// TIA Portal V17 export
// export: Created 2025-03-07T09:17:02.3863953Z, ExportSetting WithDefaults, DisplayName Totally Integrated Automation Portal, DisplayVersion V17 Update 8, DisplayName TIA Portal Openness, DisplayVersion V17 Update 8, DisplayName TIA Portal Version Control Interface, DisplayVersion V17, DisplayName SINAMICS Startdrive Advanced, DisplayVersion V17 SP2, DisplayName SINAMICS Startdrive G110M, G120, G120C, G120D, G120P, G115D, DisplayVersion V17 SP2, DisplayName SINAMICS Startdrive G130, G150, S120, S150, SINAMICS MV, S210, DisplayVersion V17 SP2, DisplayName STEP 7 Professional, DisplayVersion V17 Update 8, DisplayName SINUMERIK ONE STEP 7 Toolbox, DisplayVersion V17 Update 12, DisplayName SINUMERIK 840D sl STEP 7 Toolbox, DisplayVersion V17 Update 12, DisplayName STEP 7 Safety, DisplayVersion V17 Update 6, DisplayName WinCC Advanced, DisplayVersion V17 Update 8
DATA_BLOCK "DB7300_INTERLOCK_GENERAL"   // DB7300
{ S7_Optimized_Access := 'FALSE'; DB_Accessible_From_OPC_UA := 'FALSE' }
AUTHOR : ETXETAR
VERSION : 1.0
// stored: AutoNumber false, DBAccessibleFromOPCUA false, DBAccessibleFromWebserver true, IsOnlyStoredInLoadMemory false, IsWriteProtectedInAS false
   VAR RETAIN
      GENERAL_MACHINE : Struct
         FROM_CELL_TO_MACHINE_GENERAL : Struct
            CELL_MEAS_STA_START_CYCLE : Bool;   // CELL MEASURING STATION START CYCLE
            CELL_MEAS_STA_CALIB_CYCLE : Bool;   // CELL MEASURING STATION CALIBRATION CYCLE
            CELL_MEAS_STA_HOME_REQ : Bool;   // CELL MEASURING STATION HOME REQUEST
            CELL_MEAS_STA_FAULT : Bool;   // CELL MEASURING STATION FAULT
            CELL_MEAS_STA_RESET : Bool;   // CELL MEASURING STATION RESET
            CALIB_MODE_SLCTD_TEMP : Bool;   // CALIBRATION MODE SELECTED TEMP
            CELL_COOLING_DEGRADED_MODE : Bool;   // CELL COOLING DEGRADED MODE
            CELL_STARVED : Bool;   // CELL STARVED
            CELL_BLOCKED : Bool;   // CELL BLOCKED
         END_STRUCT;
         FROM_ROBOT_TO_UNIT_01 : Struct
            HEARTBEAT : Bool;   // ROBOT HEARTBEAT
            EMERG_STOP_OK : Bool;   // ROBOT EMERGENCY STOP OK
            ROBOT_FAULT : Bool;   // ROBOT FAULT
            SAFETY_DOOR_CLSD_LOCKD : Bool;   // ROBOT SAFETY DOOR CLOSED AND LOCKED
            CELL_EMPTY : Bool;   // ROBOT CELL EMPTY
            IN_MANUAL_MODE : Bool;   // ROBOT MANUAL MODE SELECTED
            IN_AUTO_MODE : Bool;   // ROBOT AUTO MODE SELECTED
            IN_AUTO_CYCLE_RUN : Bool;   // ROBOT CYCLE RUNNING IN AUTOMATIC MODE
            RUN_OUT_REQUEST : Bool;   // ROBOT MACHINE RUN OUT REQUEST
            RUN_OUT_COMPLETED : Bool;   // ROBOT RUN OUT COMPLETED
            SAFETY_DOOR_OPEN_REQ : Bool;   // ROBOT ANY CELL SAFETY DOOR OPEN REQUEST
            OK_TO_OPEN_SAFETY_GATES : Bool;   // OK TO OPEN SAFETY GATES
            READY_TO_SERVICE : Bool;   // ROBOT READY TO SERVICE MACHINE
            OUT_OF_COLLISION_MACHINE : Bool;   // ROBOT OUT OF COLLISION MACHINE
            OUT_OF_COLLISION_FIXTURE : Bool;   // ROBOT OUT OF COLLISION FIXTURE
            PART_ENABLED : Bool;   // ROBOT PART ENABLED
            PART_FACE_R_TO_DELIVER : Bool;   // ROBOT PART FACE R TO DELIVER IMMEDIATELY
            PART_FACE_N_TO_DELIVER : Bool;   // ROBOT PART FACE N TO DELIVER IMMEDIATELY
            OUT_OF_PARTS_FACE_R_TO_DELIVER : Bool;   // ROBOT OUT OF PARTS FACE R IN CELL TO DELIVER
            OUT_OF_PARTS_FACE_N_TO_DELIVER : Bool;   // ROBOT OUT OF PARTS FACE N IN CELL TO DELIVER
            PART_LOADED : Bool;   // ROBOT PART LOADED
            PART_UNLOADED : Bool;   // ROBOT PART UNLOADED
            FIX_SKIP_REQ : Bool;   // ROBOT FIXTURE SKIP REQUEST
            PART_TYPE_CHANGE_REQ : Bool;   // ROBOT PART TYPE CHANGE REQUEST
            PART_TYPE : Byte;   // ROBOT PART TYPE
         END_STRUCT;
         FROM_ROBOT_TO_UNIT_02 : Struct
            HEARTBEAT : Bool;   // ROBOT HEARTBEAT
            EMERG_STOP_OK : Bool;   // ROBOT EMERGENCY STOP OK
            ROBOT_FAULT : Bool;   // ROBOT FAULT
            SAFETY_DOOR_CLSD_LOCKD : Bool;   // ROBOT SAFETY DOOR CLOSED AND LOCKED
            CELL_EMPTY : Bool;   // ROBOT CELL EMPTY
            IN_MANUAL_MODE : Bool;   // ROBOT MANUAL MODE SELECTED
            IN_AUTO_MODE : Bool;   // ROBOT AUTO MODE SELECTED
            IN_AUTO_CYCLE_RUN : Bool;   // ROBOT CYCLE RUNNING IN AUTOMATIC MODE
            RUN_OUT_REQUEST : Bool;   // ROBOT MACHINE RUN OUT REQUEST
            RUN_OUT_COMPLETED : Bool;   // ROBOT RUN OUT COMPLETED
            SAFETY_DOOR_OPEN_REQ : Bool;   // ROBOT ANY CELL SAFETY DOOR OPEN REQUEST
            OK_TO_OPEN_SAFETY_GATES : Bool;   // OK TO OPEN SAFETY GATES
            READY_TO_SERVICE : Bool;   // ROBOT READY TO SERVICE MACHINE
            OUT_OF_COLLISION_MACHINE : Bool;   // ROBOT OUT OF COLLISION MACHINE
            OUT_OF_COLLISION_FIXTURE : Bool;   // ROBOT OUT OF COLLISION FIXTURE
            PART_ENABLED : Bool;   // ROBOT PART ENABLED
            PART_FACE_R_TO_DELIVER : Bool;   // ROBOT PART FACE R TO DELIVER IMMEDIATELY
            PART_FACE_N_TO_DELIVER : Bool;   // ROBOT PART FACE N TO DELIVER IMMEDIATELY
            OUT_OF_PARTS_FACE_R_TO_DELIVER : Bool;   // ROBOT OUT OF PARTS FACE R IN CELL TO DELIVER
            OUT_OF_PARTS_FACE_N_TO_DELIVER : Bool;   // ROBOT OUT OF PARTS FACE N IN CELL TO DELIVER
            PART_LOADED : Bool;   // ROBOT PART LOADED
            PART_UNLOADED : Bool;   // ROBOT PART UNLOADED
            FIX_SKIP_REQ : Bool;   // ROBOT FIXTURE SKIP REQUEST
            PART_TYPE_CHANGE_REQ : Bool;   // ROBOT PART TYPE CHANGE REQUEST
            PART_TYPE : Byte;   // ROBOT PART TYPE
         END_STRUCT;
      END_STRUCT;
      POWDER_PLC : Struct
         GENERAL : Struct
            LIFE_BIT : Bool;   // LIFE BIT
            SELECTED_ARGON_GAS : Bool;   // SELECTED ARGON GAS
            SELECTED_NITROGEN_GAS : Bool;   // SELECTED NITROGEN GAS
            SELECTED_IMPERIAL_SYSTEM : Bool;   // SELECTED IMPERIAL SYSTEM
            SELECTED_METRIC_SYSTEM : Bool;   // SELECTED METRIC SYSTEM
            POWDER_PLC_AUTO_MODE : Bool;   // POWDER PLC IN AUTO MODE
            POWDER_PLC_MAN_MODE : Bool;   // POWDER PLC IN MANUAL MODE
         END_STRUCT;
         FROM_POWDER_TO_UNIT_01 : Struct
            POWDER_UNIT_01_READY_TO_RUN : Bool;   // POWDER UNIT 01 READY TO RUN
            POWDER_UNIT_01_STOPPED : Bool;   // POWDER UNIT 01 STOPPED
            SWITCHED_ON_POWDER_UNIT_01 : Bool;   // SWITCHED ON POWDER UNIT 01
            SWITCHED_OFF_POWDER_UNIT_01 : Bool;   // SWITCHED OFF POWDER UNIT 01
            SWITCHED_ON_TEMPERATURE_JACKET_UNIT_01 : Bool;   // SWITCHED ON TEMPERATURE JACKET UNIT 01
            SWITCHED_OFF_TEMPERATURE_JACKET_UNIT_01 : Bool;   // SWITCHED OFF TEMPERATURE JACKET UNIT 01
            POWDER_UNIT_01_ALARM : Bool;   // POWDER UNIT 01 ALARM
            UNIT_01_POWDER_FEEDER_1_CARRIER_GAS_ACTUAL_LINE_1 : Real;   // UNIT 01 POWDER FEEDER 1 CARRIER GAS ACTUAL LINE 1
            UNIT_01_POWDER_FEEDER_1_DISK_SPEED_ACTUAL_LINE_1 : Real;   // UNIT 01 POWDER FEEDER 1 DISK SPEED ACTUAL LINE 1
            UNIT_01_POWDER_FEEDER_1_STIRRER_SPEED_ACTUAL_LINE_1 : Real;   // UNIT 01 POWDER FEEDER 1 STIRRER SPEED ACTUAL LINE 1
            UNIT_01_POWDER_FEEDER_1_HOPPER_TEMPERATURE_ACTUAL_LINE_1 : Real;   // UNIT 01 POWDER FEEDER 1 HOPPER TEMPERATURE ACTUAL LINE 1
            UNIT_01_POWDER_FEEDER_1_CARRIER_GAS_ACTUAL_LINE_2 : Real;   // UNIT 01 POWDER FEEDER 1 CARRIER GAS ACTUAL LINE 2
            UNIT_01_POWDER_FEEDER_1_DISK_SPEED_ACTUAL_LINE_2 : Real;   // UNIT 01 POWDER FEEDER 1 DISK SPEED ACTUAL LINE 2
            UNIT_01_POWDER_FEEDER_1_STIRRER_SPEED_ACTUAL_LINE_2 : Real;   // UNIT 01 POWDER FEEDER 1 STIRRER SPEED ACTUAL LINE 2
            UNIT_01_POWDER_FEEDER_1_HOPPER_TEMPERATURE_ACTUAL_LINE_2 : Real;   // UNIT 01 POWDER FEEDER 1 HOPPER TEMPERATURE ACTUAL LINE 2
         END_STRUCT;
         FROM_POWDER_TO_UNIT_02 : Struct
            POWDER_UNIT_02_READY_TO_RUN : Bool;   // POWDER UNIT 02 READY TO RUN
            POWDER_UNIT_02_STOPPED : Bool;   // POWDER UNIT 02 STOPPED
            SWITCHED_ON_POWDER_UNIT_02 : Bool;   // SWITCHED ON POWDER UNIT 02
            SWITCHED_OFF_POWDER_UNIT_02 : Bool;   // SWITCHED OFF POWDER UNIT 02
            SWITCHED__ON_TEMPERATURE_JACKET_UNIT_02 : Bool;   // SWITCHED ON TEMPERATURE JACKET UNIT 02
            SWITCHED_OFF_TEMPERATURE_JACKET_UNIT_02 : Bool;   // SWITCHED OFF TEMPERATURE JACKET UNIT 02
            POWDER_UNIT_02_ALARM : Bool;   // POWDER UNIT 02 ALARM
            UNIT_02_POWDER_FEEDER_1_CARRIER_GAS_ACTUAL_LINE_1 : Real;   // UNIT 02 POWDER FEEDER 1 CARRIER GAS ACTUAL LINE 1
            UNIT_02_POWDER_FEEDER_1_CARRIER_GAS_ACTUAL_LINE_2 : Real;   // UNIT 02 POWDER FEEDER 1 CARRIER GAS ACTUAL LINE 2
            UNIT_02_POWDER_FEEDER_1_DISK_SPEED_ACTUAL_LINE_1 : Real;   // UNIT 02 POWDER FEEDER 1 DISK SPEED ACTUAL LINE 1
            UNIT_02_POWDER_FEEDER_1_DISK_SPEED_ACTUAL_LINE_2 : Real;   // UNIT 02 POWDER FEEDER 1 DISK SPEED ACTUAL LINE 2
            UNIT_02_POWDER_FEEDER_1_STIRRER_SPEED_ACTUAL_LINE_1 : Real;   // UNIT 02 POWDER FEEDER 1 STIRRER SPEED ACTUAL LINE 1
            UNIT_02_POWDER_FEEDER_1_STIRRER_SPEED_ACTUAL_LINE_2 : Real;   // UNIT 02 POWDER FEEDER 1 STIRRER SPEED ACTUAL LINE 2
            UNIT_02_POWDER_FEEDER_1_HOPPER_TEMPERATURE_ACTUAL_LINE_1 : Real;   // UNIT 02 POWDER FEEDER 1 HOPPER TEMPERATURE ACTUAL LINE 1
            UNIT_02_POWDER_FEEDER_1_HOPPER_TEMPERATURE_ACTUAL_LINE_2 : Real;   // UNIT 02 POWDER FEEDER 1 HOPPER TEMPERATURE ACTUAL LINE 2
            UNIT_02_POWDER_FEEDER_2_CARRIER_GAS_ACTUAL_LINE_1 : Real;   // UNIT 02 POWDER FEEDER 2 CARRIER GAS ACTUAL LINE 1
            UNIT_02_POWDER_FEEDER_2_CARRIER_GAS_ACTUAL_LINE_2 : Real;   // UNIT 02 POWDER FEEDER 2 CARRIER GAS ACTUAL LINE 2
            UNIT_02_POWDER_FEEDER_2_DISK_SPEED_ACTUAL_LINE_1 : Real;   // UNIT 02 POWDER FEEDER 2 DISK SPEED ACTUAL LINE 1
            UNIT_02_POWDER_FEEDER_2_STIRRER_SPEED_ACTUAL_LINE_1 : Real;   // UNIT 02 POWDER FEEDER 2 STIRRER SPEED ACTUAL LINE 1
            UNIT_02_POWDER_FEEDER_2_DISK_SPEED_ACTUAL_LINE_2 : Real;   // UNIT 02 POWDER FEEDER 2 DISK SPEED ACTUAL LINE 2
            UNIT_02_POWDER_FEEDER_2_STIRRER_SPEED_ACTUAL_LINE_2 : Real;   // UNIT 02 POWDER FEEDER 2 STIRRER SPEED ACTUAL LINE 2
            UNIT_02_POWDER_FEEDER_2_HOPPER_TEMPERATURE_ACTUAL_LINE_1 : Real;   // UNIT 02 POWDER FEEDER 2 HOPPER TEMPERATURE ACTUAL LINE 1
            UNIT_02_POWDER_FEEDER_2_HOPPER_TEMPERATURE_ACTUAL_LINE_2 : Real;   // UNIT 02 POWDER FEEDER 2 HOPPER TEMPERATURE ACTUAL LINE 2
         END_STRUCT;
      END_STRUCT;
      MEASURING_STATION : Struct
         FROM_ROBOT_TO_MEAS_STATION : Struct
            HEARTBEAT : Bool;   // ROBOT HEARTBEAT
            EMERG_STOP_OK : Bool;   // ROBOT EMERGENCY STOPOK
            SAFETY_DOOR_CLSD_LOCKD : Bool;   // ROBOT SAFETY DOOR CLOSED AND LOCKED
            CELL_EMPTY : Bool;   // ROBOT CELL EMPTY
            IN_MANUAL_MODE : Bool;   // ROBOT MANUAL MODE SELECTED
            IN_AUTO_MODE : Bool;   // ROBOT AUTO MODE SELECTED
            IN_AUTO_CYCLE_RUN : Bool;   // ROBOT CYCLE RUNNING IN AUTOMATIC MODE
            IN_WARM_UP_CYCLE_RUN : Bool;   // ROBOT WARM UP CYCLE RUNNING
            RUN_OUT_REQUEST : Bool;   // ROBOT MACHINE RUN OUT REQUEST
            RUN_OUT_COMPLETED : Bool;   // ROBOT RUN OUT COMPLETED
            SAFETY_DOOR_OPEN_REQ : Bool;   // ROBOT ANY CELL SAFETY DOOR OPEN REQUEST
            READY_TO_UNLOAD : Bool;   // ROBOT READY TO UNLOAD
            READY_TO_LOAD : Bool;   // ROBOT READY TO LOAD
            OUT_OF_COLLISION_STATION : Bool;   // ROBOT OUT OF COLLISION STATION
            PART_UNLOADED : Bool;   // ROBOT PART UNLOADED
            PART_LOADED : Bool;   // ROBOT PART LOADED
            PART_TYPE_CHANGE_REQ : Bool;   // ROBOT PART TYPE CHANGE REQUEST
            PART_TYPE : Byte;   // ROBOT PART TYPE
         END_STRUCT;
      END_STRUCT;
      LOAD_UNLOAD : Struct
         UNIT_01 : "LOAD_UNLOAD_ETXETAR_ROBOT_CELL";
         UNIT_02 : "LOAD_UNLOAD_ETXETAR_ROBOT_CELL";
         UNIT_03 : "LOAD_UNLOAD_ETXETAR_ROBOT_CELL";
      END_STRUCT;
      AUX_SIGNALS_INTERFACE : Struct
         GENERAL : Struct
            "MEASURING STATION FAULT" : Bool;   // CELL MEASURING STATION FAULT
            "DEGRADED MODE FAULT" : Bool;   // CELL COOLING DEGRADED MODE FAULT
            TIMER_MEASURING_IN_PRCS : TOF_TIME;   // TIMER MEASURING IN PROCESS
            TIMER_MEASURING_DONE : TOF_TIME;   // TIMER MEASURING DONE
         END_STRUCT;
         UNIT_01 : Struct
            LIFE_BIT_FAULT : Bool;   // HEARTBEAT COMMUNICATION ALARM
            EMERGENCY_STOP_ACTIVE : Bool;   // EMERGENCY STOP ACTIVE ALARM
            ROBOT_FAULT : Bool;   // ROBOT FAULT ALARM
            FACE_R_LOAD_REQ_AUX : Bool;   // FACE R LOAD REQUEST AUX
            FACE_N_LOAD_REQ_AUX : Bool;   // FACE N LOAD REQUEST AUX
            "LIFE SING COUNTER" : CTU_INT;
         END_STRUCT;
         UNIT_02 : Struct
            LIFE_BIT_FAULT : Bool;   // HEARTBEAT COMMUNICATION ALARM
            EMERGENCY_STOP_ACTIVE : Bool;   // EMERGENCY STOP ACTIVE ALARM
            ROBOT_FAULT : Bool;   // ROBOT FAULT ALARM
            FACE_R_LOAD_REQ_AUX : Bool;   // FACE R LOAD REQUEST AUX
            FACE_N_LOAD_REQ_AUX : Bool;   // FACE N LOAD REQUEST AUX
            "LIFE SING COUNTER" : CTU_INT;
         END_STRUCT;
         POWDER_PLC : Struct
            LIFE_BIT_FAULT : Bool;   // HEARTBEAT COMMUNICATION ALARM
            "LIFE SING COUNTER" : CTU_INT;
         END_STRUCT;
         AUX_0 : Bool;   // AUXILIARY 0
         AUX_1 : Bool;   // AUXILIARY 1
         AUX_2 : Bool;   // AUXILIARY 2
         AUX_3 : Bool;   // AUXILIARY 3
         AUX_4 : Bool;   // AUXILIARY 4
         AUX_5 : Bool;   // AUXILIARY 5
         AUX_6 : Bool;   // AUXILIARY 6
         AUX_7 : Bool;   // AUXILIARY 7
         AUX_8 : Bool;   // AUXILIARY 8
         AUX_9 : Bool;   // AUXILIARY 9
         AUX_10 : Bool;   // AUXILIARY 10
         AUX_11 : Bool;   // AUXILIARY 11
         AUX_12 : Bool;   // AUXILIARY 12
         AUX_13 : Bool;   // AUXILIARY 13
         AUX_14 : Bool;   // AUXILIARY 14
         AUX_15 : Bool;   // AUXILIARY 15
      END_STRUCT;
      PART_A : Struct
         UNIT_01 : "PART_STATUS_CLADDING";
         UNIT_02 : "PART_STATUS_CLADDING";
         UNIT_03 : "PART_STATUS_CLADDING";
      END_STRUCT;
   END_VAR
BEGIN
   AUX_SIGNALS_INTERFACE.GENERAL.TIMER_MEASURING_IN_PRCS.PT := T#3s;
   AUX_SIGNALS_INTERFACE.GENERAL.TIMER_MEASURING_DONE.PT := T#3s;
END_DATA_BLOCK
